// TIA Portal project "XSFW_TIA31001_A0" (V15)

(* hardware
DEVICE "S7-1200 station_1"  S7-1200 Station
   slot 0: "Rack_0"  S7-1200 Rack  Rack  V1.0
   slot 1: "PLC_Divider"  CPU 1214C DC/DC/DC  6ES7 214-1AG40-0XB0  V4.2
   slot 2: "AI 4x13BIT/AQ 2x14BIT_1"  6ES7 234-4HE32-0XB0  V2.0
   slot 101: "CM 1243-5"  CM 1243-5  6GK7 243-5DX30-0XE0  V1.3
DEVICE "CSM"  SCALANCE X-Station
   slot 0: "Bastidor SCALANCE X"  Rail
   slot 0: "Switch"  6GK7 277-1AA00-0AA0
DEVICE "HMI_1"  KTP700 Basic PN
   slot 0: "HMI_1"  KTP700 Basic PN  6AV2 123-2GB03-0AX0  15.0.0.0
   slot 1: "HMI_RT_1"  KTP700 Basic PN  6AV2 123-2GB03-0AX0  15.0.0.0
   slot 5: "HMI_1.IE_CP_1"  PROFINET Interface  15.0.0.0
      slot 1: "Interfaz PROFINET_1"  PROFINET Interface
         slot 1: "Port_1"  Port
DEVICE "Dispositivo GSD_1"  GSD.Device.PN
   slot 0: "Rack"  Rack  V1.0
   slot 0: "V90-X"  SINAMICS V90 PN V1.0  6SL3 210-5Fxxx-xxFx  V1.00
      slot 0: "SINAMICS V90 PN V1.0"  SINAMICS V90 PN V1.0
      slot 1: "PN-IO"  PN-IO
         slot 1: "Puerto 1"  Port 1
         slot 2: "Puerto 2"  Port 2
      slot 1: "Drive"  Drive
         slot 0: "Punto de acceso a módulo"  Module Access Point
         slot 1: "sin PROFIsafe"  without PROFIsafe
   slot 2: "Telegrama estándar 3, PZD-5/9"  Standard telegram 3, PZD-5/9
DEVICE "Dispositivo GSD_2"  GSD.Device.PN
   slot 0: "Rack"  Rack  V1.0
   slot 0: "V90-Y"  SINAMICS V90 PN V1.0  6SL3 210-5Fxxx-xxFx  V1.00
      slot 0: "SINAMICS V90 PN V1.0"  SINAMICS V90 PN V1.0
      slot 1: "PN-IO"  PN-IO
         slot 1: "Puerto 1"  Port 1
         slot 2: "Puerto 2"  Port 2
      slot 1: "Drive"  Drive
         slot 0: "Punto de acceso a módulo"  Module Access Point
         slot 1: "sin PROFIsafe"  without PROFIsafe
   slot 2: "Telegrama estándar 3, PZD-5/9"  Standard telegram 3, PZD-5/9
*)

// ===== PLC "PLC_Divider"  CPU 1214C DC/DC/DC =====

VAR_GLOBAL   // PLC tag table "Tabla de variables estándar"
   "Eje_1_Impulso" AT %Q0.0 : Bool;
   "Eje_1_Sentido" AT %Q0.1 : Bool;
   "Eje_1_Drive_IN" AT %I68.0 : "PD_TEL3_IN";
   "Eje_1_Drive_OUT" AT %Q64.0 : "PD_TEL3_OUT";
   "HSC_1_Up" AT %I0.0 : Bool;
   "HSC_1_Down" AT %I0.1 : Bool;
   "Eje_Y_Drive_IN" AT %I104.0 : "PD_TEL3_IN";
   "Eje_Y_Drive_OUT" AT %Q74.0 : "PD_TEL3_OUT";
END_VAR

DATA_BLOCK "Bloque de datos_1"   // DB2
{ S7_Optimized_Access := 'TRUE' }
VERSION : 0.1
   VAR
      "a" : Bool;
   END_VAR
BEGIN
END_DATA_BLOCK

DATA_BLOCK "Eje_X"   // DB1, Motion_DB
{ S7_Optimized_Access := 'TRUE' }
AUTHOR : SIMATIC
FAMILY : BasicMC
NAME : TO_PosAx
VERSION : 6.0
// stored: InstanceOfName TO_PositioningAxis
"TO_PositioningAxis"
BEGIN
   // Axis.Encoder.TelegramAddressOutCU = %Q64.0
   // Axis.Encoder.TelegramAddressInCU = %I68.0
   // Axis.Encoder.DoNameCU = V90-X.Drive_Encóder1
   // Axis.Drive.TelegramAddressOutCU = %Q64.0
   // Axis.Drive.TelegramAddressInCU = %I68.0
   // Axis.Drive.TelegramType = 2
   // Axis.Drive.DoNameCU = V90-X.Accionamiento_1
   // Axis.LengthUnitNormalized.Time = 1
   // Axis.LengthUnitNormalized.Distance = -2
   // Axis.Encoder.SelectedHscIndexCU = -1
   // Axis.Encoder.DbTypeCU = Classic
   // Axis.Drive.DbTypeCU = Classic
END_DATA_BLOCK

DATA_BLOCK "Eje_Y"   // DB4, Motion_DB
{ S7_Optimized_Access := 'TRUE' }
AUTHOR : SIMATIC
FAMILY : BasicMC
NAME : TO_PosAx
VERSION : 6.0
// stored: InstanceOfName TO_PositioningAxis
"TO_PositioningAxis"
BEGIN
   // Axis.Encoder.TelegramAddressOutCU = %Q74.0
   // Axis.Encoder.TelegramAddressInCU = %I104.0
   // Axis.Encoder.DoNameCU = V90-Y.Drive_Encóder1
   // Axis.Drive.TelegramAddressOutCU = %Q74.0
   // Axis.Drive.TelegramAddressInCU = %I104.0
   // Axis.Drive.TelegramType = 2
   // Axis.Drive.DoNameCU = V90-Y.Drive
   // Axis.LengthUnitNormalized.Time = 1
   // Axis.LengthUnitNormalized.Distance = -2
   // Axis.Encoder.SelectedHscIndexCU = -1
   // Axis.Encoder.DbTypeCU = Classic
   // Axis.Drive.DbTypeCU = Classic
END_DATA_BLOCK

ORGANIZATION_BLOCK "Main"   // OB1, LAD, ProgramCycle
TITLE = "Main Program Sweep (Cycle)"
{ S7_Optimized_Access := 'TRUE' }
VERSION : 0.1
   VAR_INPUT
      Initial_Call : Bool;   // Initial call of this OB
      Remanence : Bool;   // =True, if remanent data are available
   END_VAR
BEGIN

REGION Network 1
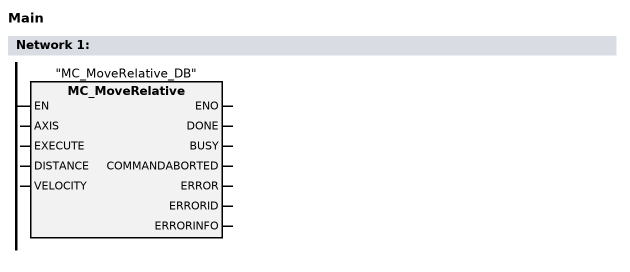
   "MC_MoveRelative_DB"();   // MC_MoveRelative
END_REGION
END_ORGANIZATION_BLOCK